(* IEC 61131-3 sources: AXOpen/src/components.siemens.identification/ctrl/src/AxoIdentificationDataTypes (part 2) *)

                                                aRxref[statLowerBoundRxref + TO_DINT(statRecvOffset) - 1] := tempZeroValue;

                                                IF statLastMoveError <> 0 THEN
                                                    tempIntError := true;
                                                    statIntStatus := DWORD#16#E7FE0400;
                                                    EXIT;
                                                END_IF;
                                            END_IF;
                                        END_IF;

                                        // check dbl // if PDU > 240, length is only in byte 0 and 1
                                        IF stHwConnect.STATIC.buf_max > UINT#240 THEN
                                            tempW.%B0   :=  stHwConnect.Static.pnConfigRecord.record.buf[1];
                                            tempW.%B1   :=  stHwConnect.Static.pnConfigRecord.record.buf[0];
                                            statSize    :=  TO_UINT(tempW);
                                        ELSE
                                            statSize := TO_UINT(stHwConnect.Static.pnConfigRecord.record.buf[10]);
                                        END_IF;
                                        IF statSize > stHwConnect.STATIC.buf_maxdata THEN
                                            // invalid data block length
                                            tempIntError := true;
                                            statIntStatus := DWORD#16#E5FE0700;
                                            EXIT;
                                        ELSIF statSize > UINT#0 AND statDbn = UINT#1 THEN
                                            // data arrived, first packet -> reset TRLEN
                                            nTrlen := 0;
                                        END_IF;

                                        IF statSize > UINT#0 THEN
                                            // recv_offset was adjusted by RXSTART
                                            tempLi := statRxbuflen - statRecvOffset;
                                            IF statSize > tempLi THEN
                                                // not enough space in buffer
                                                tempIntError := true;
                                                statIntStatus := DWORD#16#E7FE0400;
                                                EXIT;
                                            ELSE
                                                // anything ok, copy over data
                                                // MEMCPY(
                                                //     destAddr:=ADR(aRxref[statLowerBoundRxref + UDINT_TO_DINT(statRecvOffset)]) ,
                                                //     srcAddr:=ADR(stHwConnect.Static.pnConfigRecord.record.buf[stHwConnect.STATIC.buf_header]) ,
                                                //     n:=UINT_TO_UDINT(statSize));

                                                FOR i := 1 TO TO_INT(statSize) DO
                                                    aRxref[statLowerBoundRxref + TO_DINT(statRecvOffset) + TO_DINT(i) - DINT#1] := stHwConnect.Static.pnConfigRecord.record.buf[stHwConnect.STATIC.buf_header + TO_UINT(i) - UINT#1];
                                                END_FOR;

                                                // IF TypeOfElements(txref) = Char THEN
                                                //     FOR tempLoop := 0 TO statSize - 1 DO

                                                //         tempChar := BYTE_TO_CHAR(hw_connect.Static.pnConfigRecord.record.buf[hw_connect.STATIC.buf_header + tempLoop]);

                                                //         statLastMoveError := MOVE_BLK_VARIANT(SRC := tempChar,
                                                //                                             COUNT := 1,
                                                //                                             SRC_INDEX := 0,
                                                //                                             DEST_INDEX := statRecvOffset + tempLoop,
                                                //                                             DEST => rxref);
                                                //     END_FOR;
                                                // ELSE

                                                //     statLastMoveError := MOVE_BLK_VARIANT(SRC := hw_connect.STATIC.buf,
                                                //                                         COUNT := INT_TO_UDINT(statSize),
                                                //                                         SRC_INDEX := hw_connect.STATIC.buf_header,
                                                //                                         DEST_INDEX := statRecvOffset,
                                                //                                         DEST => rxref);

                                                // END_IF;
                                                // // error at mov_blk
                                                // IF statLastMoveError <> 0 THEN
                                                //     tempIntError := true;
                                                //     statIntStatus := 16#E7FE0400;
                                                //     EXIT;
                                                // END_IF;

                                                statRecvOffset := statRecvOffset + statSize;
                                                nTrlen := nTrlen + statSize;
                                                // add one to length if a zero-byte was added in buffer
                                                IF tempShift THEN
                                                    nTrlen := nTrlen + 1;
                                                    tempShift := false;
                                                END_IF;
                                            END_IF;
                                        END_IF;

                                        // read next telegram
                                        IF NOT tempFinished THEN
                                            stHwConnect.STATIC.state := STATE6;
                                        ELSE
                                            // -command- complete
                                            //Change 03.00.02

                                            // if chained commands => decrease chained counter
                                            IF statChainedCounter > UINT#1 THEN
                                                statChainedCounter := statChainedCounter - UINT#1;
                                                stHwConnect.STATIC.state := STATE6;
                                                statAdb := UINT#0;
                                                EXIT;
                                            ELSE
                                                stHwConnect.STATIC.state := STATE4;

                                                // map input RPTCMD to RPTCMD_cyc
                                                stHwConnect.STATIC.RPTCMD_cyc := bRepeatCommand;

                                                IF statChainedStatus <> DWORD#0 THEN
                                                    tempIntError := true;
                                                    EXIT;
                                                END_IF;
                                            END_IF;

                                            // set outputs
                                            bDone := TRUE;
                                            bBusy := FALSE;
                                            bError := FALSE;
                                            // reset pib-status-variables
                                            stHwConnect.STATIC.STATUS_IN_WORK := false;
                                            stHwConnect.STATIC.STATUS_INITIALISATION := false;
                                        END_IF;
                                    END_IF;
                                END_IF;
                            STATE8: //---------------------end of soft reset----------------------------
                                IF NOT stHwConnect.STATIC.SRESET_active THEN
                                    // reset command counter
                                    stHwConnect.STATIC.old_CC_H := FALSE;
                                    stHwConnect.STATIC.old_CC_L := FALSE;
                                    // remember acknowledge counter
                                    stHwConnect.STATIC.old_AC_H := stHwConnect.STATIC.AC_H;
                                    stHwConnect.STATIC.old_AC_L := stHwConnect.STATIC.AC_L;
                                    // reset chained counter
                                    statChainedCounter := UINT#1;
                                    statFixChainedCounter := UINT#1;

                                    // reset status-variables
                                    stHwConnect.STATIC.STATUS_IN_WORK := FALSE;
                                    stHwConnect.STATIC.STATUS_INITIALISATION := FALSE;
                                    // reset state-variable
                                    stHwConnect.STATIC.state := STATE4;

                                    // drop repeat
                                    stHwConnect.STATIC.RPTCMD_cyc := FALSE;
                                    bRepeatActive := FALSE;
                                    // set outputs
                                    bDone := TRUE;
                                    bBusy := FALSE;
                                    bError := FALSE;
                                    nStatus := DWORD#0;
                                END_IF;

                            ELSE
                                tempIntError := true;
                                statIntStatus := DWORD#16#E7FE0801;
                        END_CASE;
                    END_FOR;
                END_IF;

                // check for timeout of pdu_detection
                IF statPduDetection THEN
                    statTimeout(signal := TRUE,
                                duration := stHwConnect.STATIC.timeout_reset);
                    IF statTimeout.output = TRUE THEN
                        tempIntError := TRUE;
                        statIntStatus := DWORD#16#E7FE0800;
                    END_IF;
                END_IF;

                //set pn information
                stHwConnect.Static.pnConfigRecord.nApi := stHwConnect.API;
                stHwConnect.Static.pnConfigRecord.nSlot := stHwConnect.SLOT;
                stHwConnect.Static.pnConfigRecord.nSubslot := stHwConnect.SUB_SLOT;
                stHwConnect.Static.pnConfigRecord.nNrAr := stHwConnect.AR_NUMBER;
                stHwConnect.Static.pnConfigRecord.record.nIndex := TO_WORD(stHwConnect.Static.index);

                statWRREC(  id      :=  stHwConnect.HW_ID,
                            index   :=  stHwConnect.STATIC.index,
                            length  :=  TO_UINT(stHwConnect.Static.pnConfigRecord.record.nLen) + PN_CONFIGRECORD_HEADER_LEN,
                            record	:=  stHwConnect.Static.pnConfigRecord.record.buf);

                statRDREC(  id          :=  stHwConnect.HW_ID,
                            index       :=  stHwConnect.STATIC.index,
                            maxLength  :=  stHwConnect.Static.buf_max,
                            record	    :=  stHwConnect.Static.pnConfigRecord.record.buf);

                // statAdsRdWrt(
                //             NETID:= stHwConnect.AMS_NET_ID,
                //             PORT:= stHwConnect.PORT,
                //             IDXGRP:= 16#0000_F823,
                //             IDXOFFS:= 16#0000_0000,
                //             WRITELEN:= stHwConnect.Static.pnConfigRecord.record.nLen + PN_CONFIGRECORD_HEADER_LEN,
                //             READLEN:= stHwConnect.Static.pnConfigRecord.record.nLen,
                //             SRCADDR:= ADR(stHwConnect.Static.pnConfigRecord),
                //             DESTADDR:= ADR(stHwConnect.Static.pnConfigRecord.record.buf),
                //             // WRTRD:= ,
                //             TMOUT:= ADS_TIMEOUT//,
                //             // BUSY=> ,
                //             // ERR=> ,
                //             // ERRID=>
                //             );

                statEmptyCycle := FALSE;

            // save istantly rising errors for statemachine
            // statSaveAdsError := statAdsRdWrt.ERR;
            // statIntAdsErrId := statAdsRdWrt.ERRID;
            statSaveAdsError := statWRREC.error OR statRDREC.error;
            IF statWRREC.error THEN
                statIntAdsErrId := TO_UDINT(statWRREC.status);
            ELSIF statRDREC.error THEN
                statIntAdsErrId := TO_UDINT(statRDREC.status);
            ELSE
                statIntAdsErrId := UDINT#0;
            END_IF;

                // error handling
                IF tempIntError THEN
                    // if chain is not at the end don't finish the block
                    IF (statChainedCounter > UINT#16#01) AND (stHwConnect.STATIC.state > UINT#16#05) THEN
                        statChainedCounter := statChainedCounter - UINT#1;
                        stHwConnect.STATIC.state := STATE6;
                        statAdb := UINT#0;
                        // save only first error-status in a chain
                        IF statChainedStatus = DWORD#16#0 THEN
                            statChainedStatus := statIntStatus;
                        END_IF;
                        //Send all telegrams of one Command  //Change 03.00.01
                        //ELSIF tempDbn < tempAdb AND hw_connect.Static.state = STATE7 THEN //Change 03.00.05
                        //    hw_connect.Static.state := STATE6;
                    ELSE
                        // reset pib-status-variables
                        stHwConnect.STATIC.STATUS_IN_WORK := false;
                        stHwConnect.STATIC.STATUS_INITIALISATION := false;
                        tempIntError := false;
                        stHwConnect.STATIC.state := STATE4;
                        statPduDetection := false;

                        // if error occured at chain, put the first error-status out
                        IF statChainedStatus <> DWORD#16#0 THEN
                            statIntStatus := statChainedStatus;
                            statChainedStatus := DWORD#16#0;
                        END_IF;

                        // set output variables
                        bDone := FALSE;
                        bBusy := FALSE;
                        bError := TRUE;
                        nStatus := statIntStatus;

                        // save last status + timestamp
                        statLastErrorStatus := statIntStatus;

                    END_IF;
                END_IF;
                ELSE
                    statErrorCounter := statErrorCounter + 1;
                END_IF;

        END_METHOD
    END_CLASS
END_NAMESPACE

(* ---- Axo_IID_CMD_STRUCT.st ---- *)
NAMESPACE AXOpen.Components.SIEM.Identification
    {S7.extern=ReadWrite}
    CLASS Axo_IID_CMD_STRUCT
        VAR PUBLIC
            CMD			    :   eAxo_IID_COMMANDS;	                    //Command ID
            ATTRIBUTES	    :   BYTE                    :=  BYTE#16#0;	//Subcommands
            OFFSETBUFFER    :   UINT                    :=  UINT#0;     //Offset for receive buffer
            EPCID_UID	    :   ARRAY[1..62] OF BYTE;
            LEN_DATA	    :   WORD                    :=WORD#16#0;	//Length of data
            ADDR_TAG	    :   DWORD                   :=DWORD#16#0;	//physical address on tag
            CONFIG		    :   BYTE                    :=BYTE#16#0;	//Config Mode for Init
            CHAINED		    :   BOOL                    :=FALSE;		//Chained Bit: 1= chained; 0=unchained
            EXT_UHF		    :   Axo_IID_IN_EXT_UHF;	                    //further Atrributes for extended UHF commands
        END_VAR
    END_CLASS
END_NAMESPACE

(* ---- Axo_IID_HW_CONNECT.st ---- *)
NAMESPACE AXOpen.Components.SIEM.Identification

(*
+-----------+-------------------------------------------+------------------------------------------------------+---------------------+
|           |             RF61xR/RF68xR                 |                     RF1xxC/RF360R                    |   RF180C/RF170C/MV  |
| Parameter +----------+----------+----------+----------+----------+----------+----------+----------+----------+----------+----------+
|			|   CH01   |   CH02   |   CH03   |   CH04   |   CH01   |   CH02   |   CH03   |   CH04   |CM_CONFIG |   CH01   |   CH02   |
+===========+==========+==========+==========+==========+==========+==========+==========+==========+==========+==========+==========+
| API       | 16#5B00  | 16#5B00  | 16#5B00  | 16#5B00  | 16#5B00  | 16#5B00  | 16#5B00  | 16#5B00  | 16#5B00  |   16#00  |   16#00  |
+-----------+----------+----------+----------+----------+----------+----------+----------+----------+----------+----------+----------+
| SLOT      |     1    |     1    |     1    |     1    |     2    |     3    |     4    |     5    |     1    |     1    |     1    |
+-----------+----------+----------+----------+----------+----------+----------+----------+----------+----------+----------+----------+
| SUB_SLOT  |     1    |     1    |     1    |     1    |     1    |     1    |     1    |     1    |     1    |     1    |     1    |
+-----------+----------+----------+----------+----------+----------+----------+----------+----------+----------+----------+----------+
|CM_CHANNEL |     1    |     2    |     3    |     4    |     1    |     1    |     1    |     1    |     1    |     1    |     2    |
+-----------+----------+----------+----------+----------+----------+----------+----------+----------+----------+----------+----------+
*)
    {S7.extern=ReadWrite}
    CLASS Axo_IID_HW_CONNECT
        VAR PUBLIC
            HW_ID               :   WORD    :=  WORD#16#0; 			//Hardware identifier
            AR_NUMBER 			:   WORD    :=  WORD#16#0; 			//Number of AR
            API 				:   DWORD   :=  DWORD#16#0000_5B00; //API number
            SLOT 				:   WORD    :=  WORD#16#02;  		//Slot number
            SUB_SLOT 			:   WORD    :=  WORD#16#01; 		//Subslot number
            CM_CHANNEL 			:   UINT    :=  UINT#1; 		    //channel of communication module
            STATUS_WORD         :   WORD; 					        //status word cyclic data -> link to input word of device
            CONTROL_WORD        :   WORD; 					        //control word cyclic data -> link to output word of device
            Static              :   Axo_IID_IN_SYNC;
        END_VAR
    END_CLASS
END_NAMESPACE

(* ---- Axo_IID_IN_EXT_UHF.st ---- *)
NAMESPACE AXOpen.Components.Siemens.Identification

// TYPE ST_IID_IN_EXT_UHF :
//     STRUCT
    CLASS Axo_IID_IN_EXT_UHF
        VAR PUBLIC
            LEN_ID                  :   BYTE    :=  BYTE#16#0;     //Length of EPC-ID (0-62)
            MEM_BANK                :   BYTE    :=  BYTE#16#3;     //Memory bank address
            PSWD                    :   DWORD   :=  DWORD#16#0;    //Password
            EDIT_BLACKLIST_MODE     :   BYTE    :=  BYTE#16#0;     //Mode for command "edit blacklist"
            INVENTORY_DURATION      :   WORD    :=  WORD#16#0;     //Duration for command "inventory"
            INVENTORY_DUR_UNIT      :   WORD    :=  WORD#16#0;     //Duration unit for command "inventory"
            LOCK_TAG_BANK_ACTION    :   WORD    :=  WORD#16#0;     //Lock-Action for command "lock-tag-bank"
            LOCK_TAG_BANK_MASK      :   WORD    :=  WORD#16#0;     //Lock Mask for command "lock-tag-bank"
//     END_STRUCT
// END_TYPE
    END_VAR
    END_CLASS
END_NAMESPACE

(* ---- Axo_IID_IN_PN_CONFIGRECORD.st ---- *)
NAMESPACE AXOpen.Components.Siemens.Identification
    {S7.extern=ReadWrite}
    CLASS Axo_IID_IN_PN_CONFIGRECORD
        VAR PUBLIC
            nRW         :   WORD;
            nNrAr       :   WORD;
            nApi        :   DWORD;
            nSlot       :   WORD;
            nSubslot    :   WORD;
            record      :   Axo_IID_IN_PN_RECORDDATA ;
        END_VAR
    END_CLASS
END_NAMESPACE

(* ---- Axo_IID_IN_PN_RECORDDATA.st ---- *)
NAMESPACE AXOpen.Components.Siemens.Identification

// TYPE ST_IID_IN_PN_RECORDDATA :
//     STRUCT
    CLASS Axo_IID_IN_PN_RECORDDATA
        VAR PUBLIC
            nIndex      :   WORD;
            nLen        :   WORD;
            nTrans      :   WORD;
            nReserve    :   WORD;
            buf         :   ARRAY[0..1034] OF BYTE;
//     END_STRUCT
// END_TYPE
    END_VAR
    END_CLASS
END_NAMESPACE

(* ---- Axo_IID_IN_SYNC.st ---- *)
NAMESPACE AXOpen.Components.SIEM.Identification
    {S7.extern=ReadWrite}
    CLASS Axo_IID_IN_SYNC
        VAR PUBLIC
            STATUS_IN_WORK              :   BOOL    :=  FALSE;      //command is in work
            STATUS_INITIALISATION       :   BOOL    :=  FALSE;      //initialisation is in work
            STATUS_LAST_CMD_INIT        :   BOOL    :=  FALSE;      //flag for initialisation
            sreset_request              :   BOOL    :=  FALSE;      //show that one app is in sreset
            acyc_active                 :   BOOL    :=  FALSE;      //acyc service is running
            reset_request               :   BOOL    :=  FALSE;      //shows that one reset-instruction is wait for ends of acyclic commands
            AC_H                        :   BOOL    :=  FALSE;      //ack counter high
            AC_L                        :   BOOL    :=  FALSE;      //ack counter low
            CC_H                        :   BOOL    :=  FALSE;      //cmd counter high
            CC_L                        :   BOOL    :=  FALSE;      //cmd counter low
            old_CC_H                    :   BOOL    :=  FALSE;      //previous ack counter high
            old_CC_L                    :   BOOL    :=  FALSE;      //previous ack counter low
            old_AC_H                    :   BOOL    :=  FALSE;      //previous cmd counter high
            old_AC_L                    :   BOOL    :=  FALSE;      //previous cmd counter low
            cyc_control                 :   WORD    :=  WORD#16#0;  //cyclic control word
            cyc_status                  :   WORD    :=  WORD#16#0;  //cyclic status word
            SRESET_active               :   BOOL    :=  FALSE;      //sreset active bit (cyc status word)
            SRESET_cyc                  :   BOOL    :=  FALSE;      //sreset control bit (cyc control word)
            RPTCMD_cyc                  :   BOOL    :=  FALSE;      //repeat control bit (cyc control word)
            RPTCMD_active               :   BOOL    :=  FALSE;      //repeat active bit (cyc status word)
            INIT_cyc                    :   BOOL    :=  FALSE;      //init control bit (cyc control word)
            init_active                 :   BOOL    :=  FALSE;      //init status bit (cyc status word)
            presence                    :   BOOL    :=  FALSE;      //presence-bit
            buf_header                  :   UINT    :=  UINT#11;    //length pib-header
            sequence_number             :   UINT    :=  UINT#0;     //sequence number (pib-header)
            config_value                :   BYTE    :=  BYTE#16#4;  //config mode for pdu-detection
            offset                      :   UINT    :=  UINT#0;     //offset for cyclic status/control word
            index                       :   UINT    :=  UINT#0;     //index for WRREC/RDREC
            buf_max                     :   UINT    :=  UINT#240;   //acyclic datagram buffer size
            instruction_set             :   BOOL    :=  FALSE;      //state for instruction set (1=RF68xR; 0=old CMs)
            index_set                   :   BOOL    :=  TRUE;       //state for DS-index (1=PROFINET; 0=PROFIBUS)
            timeout_repeat              :   TIME    :=  T#5S;       //timeout for repeat
            timeout_reset               :   TIME    :=  T#1M;       //timeout for init
            state                       :   UINT    :=  UINT#0;     //variable for statemachine
            buf_maxdata                 :   UINT    :=  UINT#229;   //user data size
            //buf:ARRAY[0..1034] OF BYTE;
            pnConfigRecord : Axo_IID_IN_PN_CONFIGRECORD;
        END_VAR
    END_CLASS
END_NAMESPACE

(* ---- AxoByteArray16.st ---- *)
NAMESPACE AXOpen.Components.SIEM.Identification
    {S7.extern=ReadWrite}
    CLASS PUBLIC AxoByteArray16 EXTENDS AXOpen.Core.AxoByteArray
        VAR PUBLIC
            Data : ARRAY [0..15] OF BYTE;
        END_VAR
    END_CLASS
END_NAMESPACE

(* ---- AxoData256.st ---- *)
NAMESPACE AXOpen.Components.SIEM.Identification
    {S7.extern=ReadWrite}
    CLASS PUBLIC AxoData256 EXTENDS AXOpen.Core.AxoByteArray
        VAR PUBLIC
            Data : ARRAY [0..255] OF BYTE;
        END_VAR
    END_CLASS
END_NAMESPACE
